PROGRAM MAIN
VAR
	stErrors : ST_ErrorStates; // Triggered error states
	fbErrorTriggers : FB_ErrorTriggers; // Brand new errors this cycl
    
    {attribute 'pytmc' := 'pv: @(BASE):FTL:VALVE:MANUAL_LATCH'}
    bManualValveLatch : BOOL := FALSE; //Manual latch for valves
    
    {attribute 'pytmc' := 'pv: @(BASE):FTL:LEAK'}
    fbLeakMonitor : FB_LeakMonitor; //Leak detection
    
    (*
    {attribute 'pytmc' := 'pv: @(BASE):FTL:PLC'}
	fbDiag : FB_EcatDiag; // Ethercat diagnostic
    *)
END_VAR

(*
(* Check PLC hardware for failures *)
fbDiag(AMSNetId := GVL_PLC.AMSNetId);
stErrors.bHardwareFailure := fbDiag.bError;
*)

(* Monitor for leaks on cooling loop*)
fbLeakMonitor(
    bLeakRelay01 := GVL_IO.bLeakRelay01,
    bLeakRelay02 := GVL_IO.bLeakRelay02,
    bError => stErrors.bLeakDetected
);

(* Open NC chiller loop valves if interlock logic passes *)
GVL_IO.bChillerValve01 := F_ChillerValveEnable(stErrors := stErrors) AND NOT bManualValveLatch;
GVL_IO.bChillerValve02 := F_ChillerValveEnable(stErrors := stErrors) AND NOT bManualValveLatch;

(* Check for rising-edge errors *)
fbErrorTriggers(stErrors := stErrors);

(* Check for new leak errors *)
IF fbErrorTriggers.NewLeakError() THEN
    bManualValveLatch := TRUE; //set manual latch for valves
ELSIF NOT bManualValveLatch THEN
	// If there are no new errors and manual latch is disabled, reset the errors
	fbLeakMonitor.Reset();
	fbErrorTriggers.ResetLeakTriggers();
END_IF

END_PROGRAM

(* stored: Version 1.1.0.1, ProductVersion 3.1.4022.18
   POU MAIN: Id {002ad0c3-72fa-47bb-80c4-f9448f2d52a7}, SpecialFunc None *)
